BUSY:
	IF XpFeedback[i].sName.CallMoveX.Done THEN
		seqMoveXM[i]:=DONE;
	ELSIF Xpfeedback[i].sName.CallMoveX.Aborted THEN
		seqMoveXM[i]:=ABORT;
	ELSIF Xpfeedback[i].sName.CallMoveX.Error THEN	
		seqMoveXM[i]:=ERROR;
	END_IF

DONE:
	IF NOT MoveXM[i] THEN
	   seqMoveXM[i]:=READY;
	END_IF

ERROR:
	IF NOT MoveXM[i] THEN
	   seqMoveXM[i]:=READY;
	END_IF

ABORT:
	IF NOT MoveXM[i] THEN
	   seqMoveXM[i]:=READY;
	END_IF
	
END_CASE
END_ACTION

ACTION callMoveX_2m:
//MoveX2m
(*
	CASE seqMoveX_2m OF
		INIT:
        seqMoveX_2m:=READY;	
	 READY:
	 IF MoveX_2m THEN
	ConstraintXY[i].SetValuesVADJ(V:=velocity_xy[i] , A:=15000 , D:=15000 , J:=100000 );
	 
		Xpmover[i].MoveX(commandFeedback:=xpFeedback[i][14] , targetPosition:= positionTargetX[i] , refSys:=Xpmover[i].MCTOPLC.SET.PhysicalAreaID , 
         constraint:=ConstraintXY[i] );
		seqMoveX_2m:=BUSY;
		
		Xpmover[i].MoveX(commandFeedback:=xpFeedback[i][14], targetPosition:= positionTargetX[i] , refSys:=Xpmover[i].MCTOPLC.SET.PhysicalAreaID , 
         constraint:=ConstraintXY[i] );
		seqMoveX_2m:=BUSY;
		
		
		END_IF
		
		
		
   BUSY:
    IF  XpFeedback[0][14].Done THEN
		seqMoveX_2m:=DONE;
    ELSIF Xpfeedback[0][14].Aborted THEN
		seqMoveX_2m:=ABORT;
	ELSIF Xpfeedback[0][14].Error THEN	
		seqMoveX_2m:=ERROR;
	END_IF
		//
	
		DONE:
		IF NOT MoveX_2m THEN
	       seqMoveX_2m:=READY;
		END_IF
		
		ERROR:
		IF NOT MoveX_2m THEN
	       seqMoveX_2m:=READY;
		END_IF
		
		ABORT:
		IF NOT MoveX_2m THEN
	       seqMoveX_2m:=READY;
		END_IF
		
	END_CASE
	*)
END_ACTION

ACTION callMoveY:
CASE seqMoveYM[i] OF

INIT:
	seqMoveYM[i]:=READY;	

READY:
	IF MoveYM[i]THEN
		MoveYM[i] := FALSE;
		ConstraintXY[i].SetValuesVADJ(
			V:=velocity_xy[i] ,A:=15000 , D:=15000 , J:=100000 );
	 
		Xpmover[i].MoveY(
			commandFeedback:=xpFeedback[i].sName.CallMoveY,
			targetPosition:= positionTargetY[i],
			refSys:=Xpmover[i].MCTOPLC.SET.PhysicalAreaID, 
			constraint:=ConstraintXY[i] );
		seqMoveYM[i]:=BUSY;
	END_IF
	
BUSY:
	IF XpFeedback[i].sName.CallMoveY.Done THEN
		seqMoveYM[i]:=DONE;
	ELSIF Xpfeedback[i].sName.CallMoveY.Aborted THEN
		seqMoveYM[i]:=ABORT;
	ELSIF Xpfeedback[i].sName.CallMoveY.Error THEN	
		seqMoveYM[i]:=ERROR;
	END_IF

DONE:
	IF NOT MoveYM[i] THEN
	   seqMoveYM[i]:=READY;
	END_IF

ERROR:
	IF NOT MoveYM[i] THEN
	   seqMoveYM[i]:=READY;
	END_IF

ABORT:
	IF NOT MoveYM[i] THEN
	   seqMoveYM[i]:=READY;
	END_IF
	
END_CASE
END_ACTION

ACTION callMoveZ:
CASE seqMoveZM[i] OF

INIT:
	seqMoveZM[i]:=READY;
	Constratint_ZABC[i].SetLimit(
		Coordinate:= Coord_Mcs_A1, 
		V:= 100 , 
		A:= 100 , 
		D:= 100, 
		J:= 1000);
	
READY:
	IF moveZM[i]THEN
		MoveZM[i] := FALSE;	
		Constratint_ZABC[i].AddLimit(
			Coordinate:= Coord_Mcs_A1, 
			V:= 100 , 
			A:= 100 , 
			D:= 100, 
			J:= 1000);
		Xpmover[i].MoveZ(
			commandFeedback:=xpFeedback[i].sName.CallMoveZ , 
			targetPosition:=positionTargetZ[i] , 
			constraint:=ConstraTINT_zabc[i]);
		seqMoveZM[i]:=BUSY;
	END_IF
		
BUSY:
    IF XpFeedback[i].sName.CallMoveZ.Done THEN
		seqMoveZM[i]:=DONE;
    ELSIF Xpfeedback[i].sName.CallMoveZ.Aborted THEN
		seqMoveZM[i]:=ABORT;
	ELSIF Xpfeedback[i].sName.CallMoveZ.Error THEN	
		seqMoveZM[i]:=ERROR;
	END_IF
	
DONE:
	IF NOT MoveZM[i] THEN
	   seqMoveZM[i]:=READY;
	END_IF
	
ERROR:
	IF NOT MoveZM[i] THEN
	   seqMoveZM[i]:=READY;
	END_IF
	
ABORT:
	IF NOT MoveZM[i] THEN
	   seqMoveZM[i]:=READY;
	END_IF
		
END_CASE
END_ACTION

ACTION CallReset:
CASE seqResetM[i] OF
	
INIT:
	seqResetM[i]:=READY;

READY:
	IF ResetM[i]THEN
		Xpmover[i].Reset(commandFeedback:=XpFeedBack[i].sName.CallReset);
		seqResetM[i]:=BUSY;
	END_IF
		
BUSY:
	IF xpFeedback[i].sName.CallReset.Done THEN
		ResetM[i]:=FALSE;
		seqResetM[i]:=DONE;
	END_IF
		
DONE:
	IF NOT ResetM[i] THEN
		seqResetM[i]:=READY;
	END_IF

END_CASE
END_ACTION

ACTION seq_JoinTrack:
IF bJoinTrackseq THEN
	bJoinTrackseq := FALSE;
	
	FOR i:=0 TO gvl.MAX_MOVER DO
		ConstraintXY[i].SetValuesVADJ(V:=velocity_xy[i] , A:=15000 , D:=15000 , J:=100000 );
		velocity_xy[i] := 50;
	END_FOR
	
	Xpmover[0].JoinTrack(commandFeedback:= Xpfeedback[0].sName.SeqJoinTrack,
		targetTrack:= XpTrack[E_TrackName.Wait],
		constraint := ConstraintXY[0],
		options := 0);
		
	xpmover[1].JoinTrack(commandFeedback:= Xpfeedback[1].sName.SeqJoinTrack,
		targetTrack:= XpTrack[E_TrackName.EndA],
		constraint := ConstraintXY[1],
		options := 0);
END_IF

IF bMoveTrackSeq THEN
	bMoveTrackSeq := FALSE;
	fbStateTrack[0].bMoveState := TRUE;
	fbStateTrack[1].bMoveState := TRUE;
ELSE
	fbStateTrack[0].bMoveState := FALSE;
	fbStateTrack[1].bMoveState := FALSE;
END_IF

IF GVL.bfill THEN
	GVL.bfill  := FALSE;
END_IF

diCountSum := 0;
FOR i:=0 TO GVL.MAX_MOVER DO
	diCountSum := diCountSum + fbStateTrack[i].icount;
END_FOR

IF CountReset THEN
	CountReset := FALSE;
	FOR i:=0 TO GVL.MAX_MOVER DO
		fbStateTrack[i].breset := TRUE;
	END_FOR
END_IF
END_ACTION

ACTION update:
FOR i:=0 TO gvl.MAX_MOVER DO //xpmover 
	XpMover[i].update();
	FOR k:=0 TO MAX_FEEDBACK DO	
		Xpfeedback[i].aArray[k].Update();
	END_FOR
END_FOR

FOR t:=0 TO MAX_TRACK DO
    XpTrack[t].Update();
END_FOR
END_ACTION

END_PROGRAM

// ---- GlobalTextList.TcGTLO
TEXTLIST GlobalTextList
  582 = '%0,1f'
  833 = '%0.1f'
  192 = '%0.1f /s'
  27 = '%0.1f deg/s'
  12 = '%0.1f mm/s'
  142 = '%d'
  807 = '%S'
  450 = '1'
  857 = '2'
  13 = '22'
  974 = 'A'
  287 = 'A(Rx)'
  255 = 'B'
  85 = 'B(Ry)'
  421 = 'BFILL'
  484 = 'bstop'
  865 = 'C'
  567 = 'C(Rz)'
  424 = 'count'
  375 = 'disable'
  989 = 'Disable'
  74 = 'Enable'
  644 = 'Halt'
  595 = 'JoinTrack'
  973 = 'JoinTrack\nMover2台順次'
  117 = 'JoinTrack 1'
  83 = 'LeaveTrack'
  545 = 'moveA'
  66 = 'moveB'
  980 = 'moveC'
  981 = 'MoveOn'
  361 = 'MoveOnTrack'
  549 = 'MoveOnTrack 1'
  885 = 'Mover1'
  533 = 'Mover2'
  882 = 'Mover3'
  44 = 'Mover4'
  602 = 'MoverX1'
  542 = 'MoverX2'
  668 = 'MoveTrack\nMover2台同時'
  734 = 'movex'
  52 = 'movex1'
  608 = 'movey'
  742 = 'moveY'
  360 = 'moveY1'
  884 = 'moveZ'
  86 = 'Point to Move'
  994 = 'RealTime'
  474 = 'Reset'
  187 = 'reset'
  233 = 'Target Pos'
  977 = 'velo'
  587 = 'velocity_c'
  520 = 'velocity_xy'
  226 = 'X'
  493 = 'X1'
  377 = 'Y'
  645 = 'Y1'
  95 = 'Z'
  372 = '[0]'
  901 = '[0][0]'
  862 = '[1]'
END_TEXTLIST

// ---- VISUs/Visualization.TcVIS
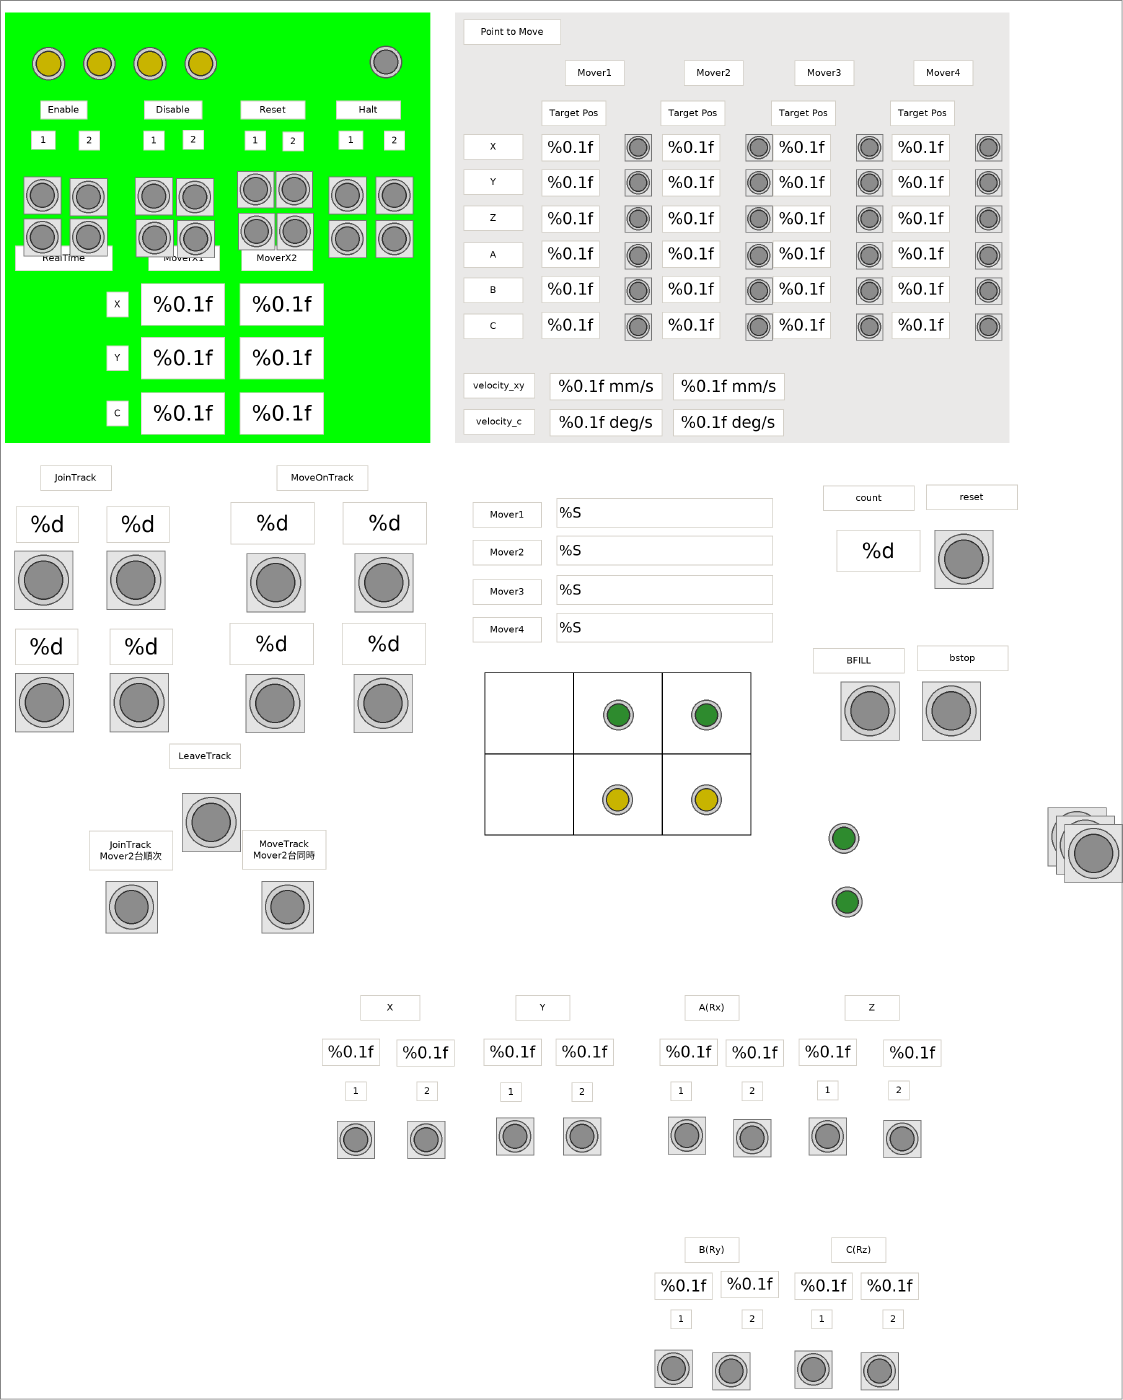
VISUALIZATION Visualization  // 1340x1670
    Rectangle (543,15 661x513)
    Rectangle (6,15 507x513)
    PushSwitch (161,194 45x80), tooltip "disable", variable: MAIN.disableM[0], behaviour: TAP, style: Switch-PushSwitch-Gray
    Lamp1 (35,43 46x66), variable: MAIN.bMoverEnable[0], style: Lamp-Lamp1-Yellow
    PushSwitchLed (402,1325 45x69), tooltip "movex", variable: MAIN.moveXM[0], behaviour: TOGGLE, style: Switch-PushSwitchLed-Gray
    Textfield (384,1239 69x32), "%0.1f", text variable: MAIN.positionTargetX[0]
        OnMouseClick: write the text variable via Default, min 60, max 660
    Textfield (430,1187 71x30), "X"
    Textfield (577,1239 69x32), "%0.1f", text variable: MAIN.positionTargetY[0]
        OnMouseClick: write the text variable via Default, min 60, max 420
    Textfield (615,1187 65x30), "Y"
    PushSwitchLed (592,1324 45x63), tooltip "moveY", variable: MAIN.moveYM[0], behaviour: TOGGLE, style: Switch-PushSwitchLed-Gray
    Textfield (553,445 85x30), "velocity_xy"
    Textfield (817,1187 65x30), "A(Rx)"
    Textfield (787,1239 69x32), "%0.1f", text variable: MAIN.positionTargetA[0]
        OnMouseClick: write the text variable via Default, min -5, max 5
    PushSwitchLed (797,1323 45x63), tooltip "moveA", variable: MAIN.moveAM[0], behaviour: TOGGLE, style: Switch-PushSwitchLed-Gray
    Textfield (817,1476 65x30), "B(Ry)"
    Textfield (781,1518 69x32), "%0.1f", text variable: MAIN.positionTargetB[0]
        OnMouseClick: write the text variable via Default, min -5, max 5
    PushSwitchLed (781,1598 45x69), tooltip "moveB", variable: MAIN.moveBM[0], behaviour: TOGGLE, style: Switch-PushSwitchLed-Gray
    Textfield (1008,1187 65x30), "Z"
    Textfield (953,1239 69x32), "%0.1f", text variable: MAIN.positionTargetZ[0]
        OnMouseClick: write the text variable via Default, min 2, max 5
    PushSwitchLed (965,1324 45x63), tooltip "moveZ", variable: MAIN.moveZM[0], behaviour: TOGGLE, style: Switch-PushSwitchLed-Gray
    Textfield (992,1476 65x30), "C(Rz)"
    Textfield (948,1518 69x32), "%0.1f", text variable: MAIN.positionTargetC[0]
        OnMouseClick: write the text variable via Default
    PushSwitchLed (948,1599 45x69), tooltip "moveC", variable: MAIN.moveCM[0], behaviour: TOGGLE, style: Switch-PushSwitchLed-Gray
    Textfield (553,488 85x30), "velocity_c"
    Textfield (168,338 100x50), "%0.1f", text variable: MAIN.Xpmover[0].MCTOPLC.ACT.ActPos.x
    Textfield (168,402 100x50), "%0.1f", text variable: MAIN.Xpmover[0].MCTOPLC.ACT.ActPos.y
    Textfield (168,468 100x50), "%0.1f", text variable: MAIN.Xpmover[0].MCTOPLC.ACT.ActPos.c
    Textfield (177,293 85x30), "MoverX1"
    PushSwitch (17,657 70x70), variable: MAIN.JoinTrack[0], behaviour: TOGGLE, style: Switch-PushSwitch-Gray
    PushSwitch (217,946 70x70), variable: MAIN.LeaveTrack[0], behaviour: TOGGLE, style: Switch-PushSwitch-Gray
    Textfield (48,555 85x30), "JoinTrack"
    Textfield (202,887 85x30), "LeaveTrack"
    Textfield (19,604 75x43), "%d", text variable: MAIN.numberTrack[0]
        OnMouseClick: write the text variable via Default, min 0
    PushSwitch (283,195 44x62), variable: MAIN.ResetM[0], invisible if: MAIN.ResetM, behaviour: TOGGLE, style: Switch-PushSwitch-Gray
    Textfield (48,120 56x22), "Enable"
    Textfield (172,120 69x22), "Disable"
    Textfield (287,120 77x22), "Reset"
    PushSwitch (392,193 45x80), variable: MAIN.HaltM[0], invisible if: MAIN.HaltM, behaviour: TOGGLE, style: Switch-PushSwitch-Gray
    Textfield (37,156 29x22), "1"
    Textfield (94,156 25x23), "2"
    Lamp1 (96,44 45x64), variable: MAIN.bMoverEnable[1], style: Lamp-Lamp1-Yellow
    Textfield (171,156 25x23), "1"
    Textfield (218,155 25x23), "2"
    PushSwitch (210,195 45x80), tooltip "disable", variable: MAIN.disableM[1], behaviour: TAP, style: Switch-PushSwitch-Gray
    Textfield (292,156 25x23), "1"
    PushSwitch (329,195 44x62), variable: MAIN.ResetM[1], invisible if: MAIN.ResetM, behaviour: TOGGLE, style: Switch-PushSwitch-Gray
    Textfield (337,157 25x23), "2"
    Textfield (497,1290 25x23), "2"
    Textfield (412,1290 25x23), "1"
    PushSwitchLed (486,1325 45x69), tooltip "movex", variable: MAIN.moveXM[1], behaviour: TOGGLE, style: Switch-PushSwitchLed-Gray
    Textfield (473,1240 69x32), "%0.1f", text variable: MAIN.positionTargetX[1]
        OnMouseClick: write the text variable via Default, min 60, max 660
    Textfield (663,1239 69x32), "%0.1f", text variable: MAIN.positionTargetY[1]
        OnMouseClick: write the text variable via Default, min 60, max 420
    PushSwitchLed (672,1324 45x63), tooltip "moveY", variable: MAIN.moveYM[1], behaviour: TOGGLE, style: Switch-PushSwitchLed-Gray
    Textfield (866,1240 69x32), "%0.1f", text variable: MAIN.positionTargetA[1]
        OnMouseClick: write the text variable via Default, min -5, max 5
    PushSwitchLed (875,1326 45x63), tooltip "moveA", variable: MAIN.moveAM[1], behaviour: TOGGLE, style: Switch-PushSwitchLed-Gray
    PushSwitchLed (1054,1327 45x63), tooltip "moveZ", variable: MAIN.moveZM[1], behaviour: TOGGLE, style: Switch-PushSwitchLed-Gray
    Textfield (1054,1240 69x32), "%0.1f", text variable: MAIN.positionTargetZ[1]
        OnMouseClick: write the text variable via Default, min 2, max 5
    PushSwitchLed (850,1601 45x69), tooltip "moveB", variable: MAIN.moveBM[1], behaviour: TOGGLE, style: Switch-PushSwitchLed-Gray
    Textfield (860,1516 69x32), "%0.1f", text variable: MAIN.positionTargetB[0]
        OnMouseClick: write the text variable via Default, min -5, max 5
    Textfield (1027,1518 69x32), "%0.1f", text variable: MAIN.positionTargetC[1]
        OnMouseClick: write the text variable via Default
    PushSwitchLed (1027,1601 45x69), tooltip "moveC", variable: MAIN.moveCM[1], behaviour: TOGGLE, style: Switch-PushSwitchLed-Gray
    Textfield (288,293 85x30), "MoverX2"
    Textfield (286,338 100x50), "%0.1f", text variable: MAIN.Xpmover[1].MCTOPLC.ACT.ActPos.x
    Textfield (286,402 100x50), "%0.1f", text variable: MAIN.Xpmover[1].MCTOPLC.ACT.ActPos.y
    Textfield (286,468 100x50), "%0.1f", text variable: MAIN.Xpmover[1].MCTOPLC.ACT.ActPos.c
    PushSwitch (448,193 45x80), variable: MAIN.HaltM[1], invisible if: MAIN.HaltM, behaviour: TOGGLE, style: Switch-PushSwitch-Gray
    Textfield (404,156 29x22), "1"
    Textfield (458,156 25x23), "2"
    Textfield (597,1291 25x23), "1"
    Textfield (682,1291 25x23), "2"
    Textfield (800,1290 25x23), "1"
    Textfield (885,1290 25x23), "2"
    Textfield (975,1289 25x23), "1"
    Textfield (1060,1289 25x23), "2"
    Textfield (800,1562 25x23), "1"
    Textfield (885,1562 25x23), "2"
    Textfield (968,1562 25x23), "1"
    Textfield (1053,1562 25x23), "2"
    Textfield (553,160 71x30), "X"
    Textfield (674,72 71x30), "Mover1"
    Textfield (646,160 69x32), "%0.1f", text variable: MAIN.positionTargetX[0]
        OnMouseClick: write the text variable via Default, min 60, max 660
    PushSwitch (731,160 61x32), variable: MAIN.moveXM[0], behaviour: TOGGLE, style: Switch-PushSwitch-Gray
    Textfield (553,202 71x30), "Y"
    Textfield (646,202 69x32), "%0.1f", text variable: MAIN.positionTargetY[0]
        OnMouseClick: write the text variable via Default, min 60, max 420
    PushSwitch (731,202 61x32), variable: MAIN.moveYM[0], behaviour: TOGGLE, style: Switch-PushSwitch-Gray
    Textfield (553,245 71x30), "Z"
    Textfield (646,245 69x32), "%0.1f", text variable: MAIN.positionTargetZ[0]
        OnMouseClick: write the text variable via Default, min 2, max 5
    PushSwitch (731,245 61x32), variable: MAIN.moveZM[0], behaviour: TOGGLE, style: Switch-PushSwitch-Gray
    Textfield (553,289 71x30), "A"
    PushSwitch (731,289 61x32), variable: MAIN.moveAM[0], behaviour: TOGGLE, style: Switch-PushSwitch-Gray
    Textfield (553,331 71x30), "B"
    PushSwitch (731,331 61x32), variable: MAIN.moveBM[0], behaviour: TOGGLE, style: Switch-PushSwitch-Gray
    Textfield (553,374 71x30), "C"
    PushSwitch (731,374 61x32), variable: MAIN.moveCM[0], behaviour: TOGGLE, style: Switch-PushSwitch-Gray
    Textfield (646,287 69x32), "%0.1f", text variable: MAIN.positionTargetA[0]
        OnMouseClick: write the text variable via Default, min -5, max 5
    Textfield (646,329 69x32), "%0.1f", text variable: MAIN.positionTargetB[0]
        OnMouseClick: write the text variable via Default, min -5, max 5
    Textfield (646,372 69x32), "%0.1f", text variable: MAIN.positionTargetC[0]
        OnMouseClick: write the text variable via Default
    Textfield (816,72 71x30), "Mover2"
    Textfield (790,160 69x32), "%0.1f", text variable: MAIN.positionTargetX[1]
        OnMouseClick: write the text variable via Default, min 60, max 660
    PushSwitch (875,160 61x32), variable: MAIN.moveXM[1], behaviour: TOGGLE, style: Switch-PushSwitch-Gray
    Textfield (790,202 69x32), "%0.1f", text variable: MAIN.positionTargetY[1]
        OnMouseClick: write the text variable via Default, min 60, max 420
    PushSwitch (875,202 61x32), variable: MAIN.moveYM[1], behaviour: TOGGLE, style: Switch-PushSwitch-Gray
    Textfield (790,245 69x32), "%0.1f", text variable: MAIN.positionTargetZ[1]
        OnMouseClick: write the text variable via Default, min 2, max 5
    PushSwitch (875,245 61x32), variable: MAIN.moveZM[1], behaviour: TOGGLE, style: Switch-PushSwitch-Gray
    PushSwitch (875,289 61x32), variable: MAIN.moveAM[1], behaviour: TOGGLE, style: Switch-PushSwitch-Gray
    PushSwitch (875,331 61x32), variable: MAIN.moveBM[1], behaviour: TOGGLE, style: Switch-PushSwitch-Gray
    PushSwitch (875,374 61x32), variable: MAIN.moveCM[1], behaviour: TOGGLE, style: Switch-PushSwitch-Gray
    Textfield (790,287 69x32), "%0.1f", text variable: MAIN.positionTargetA[1]
        OnMouseClick: write the text variable via Default, min -5, max 5
    Textfield (790,329 69x32), "%0.1f", text variable: MAIN.positionTargetB[1]
        OnMouseClick: write the text variable via Default, min -5, max 5
    Textfield (790,372 69x32), "%0.1f", text variable: MAIN.positionTargetC[1]
        OnMouseClick: write the text variable via Default
    Textfield (646,120 77x30), "Target Pos"
    Textfield (788,120 77x30), "Target Pos"
    Textfield (553,23 116x30), "Point to Move"
    Textfield (127,348 26x30), "X"
    Textfield (127,412 26x30), "Y"
    Textfield (127,478 26x30), "C"
    Textfield (401,120 77x22), "Halt"
    Textfield (18,293 116x30), "RealTime"
    Textfield (803,445 133x32), "%0.1f mm/s", text variable: MAIN.velocity_xy[1]
        OnMouseClick: write the text variable via Default
    Textfield (656,445 134x32), "%0.1f mm/s", text variable: MAIN.velocity_xy[0]
        OnMouseClick: write the text variable via Default
    Textfield (656,488 134x32), "%0.1f deg/s", text variable: MAIN.velocity_c[0]
        OnMouseClick: write the text variable via Default
    Textfield (803,488 132x32), "%0.1f deg/s", text variable: MAIN.velocity_c[1]
        OnMouseClick: write the text variable via Default
    PushSwitch (28,193 45x80), tooltip "Enable", variable: MAIN.enableM[0], behaviour: TAP, style: Switch-PushSwitch-Gray
    PushSwitch (83,195 45x80), tooltip "Enable", variable: MAIN.enableM[1], behaviour: TAP, style: Switch-PushSwitch-Gray
    PushSwitch (294,660 70x70), variable: MAIN.fbStateTrack[0].bMoveState, behaviour: TOGGLE, style: Switch-PushSwitch-Gray
    Textfield (275,599 100x50), "%d", text variable: MAIN.fbStateTrack[0].iStateTrack
    PushSwitch (423,660 70x70), variable: MAIN.fbStateTrack[1].bMoveState, behaviour: TOGGLE, style: Switch-PushSwitch-Gray
    Textfield (409,599 100x50), "%d", text variable: MAIN.fbStateTrack[1].iStateTrack
    PushSwitch (127,657 70x70), variable: MAIN.JoinTrack[1], behaviour: TOGGLE, style: Switch-PushSwitch-Gray
    Group (578,802 318x194)
        Rectangle (0,0 106x97)
        Rectangle (0,97 106x97)
        Rectangle (106,0 106x97)
        Rectangle (106,97 106x97)
        Rectangle (212,0 106x97)
        Rectangle (212,97 106x97)
    Lamp1 (715,933 44x42), variable: GVL.bBusyB, style: Lamp-Lamp1-Yellow
    Lamp1 (821,933 44x42), variable: GVL.bBusyA, style: Lamp-Lamp1-Yellow
    Textfield (664,594 258x35), "%S", text list: 'TextList_TrackState', text index: MAIN.fbStateTrack[0].iStateTrack
    Textfield (664,639 258x35), "%S", text list: 'TextList_TrackState', text index: MAIN.fbStateTrack[1].iStateTrack
    Textfield (564,599 82x30), "Mover1"
    Textfield (564,644 82x30), "Mover2"
    PushSwitch (126,1047 62x70), variable: MAIN.bJoinTrackseq, behaviour: TOGGLE, style: Switch-PushSwitch-Gray
    Textfield (106,991 100x47), "JoinTrack Mover2台順次"
    PushSwitch (312,1047 62x70), variable: MAIN.bJoinTrackseq, behaviour: TOGGLE, style: Switch-PushSwitch-Gray
    Textfield (289,990 100x47), "MoveTrack Mover2台同時"
    Textfield (330,555 109x30), "MoveOnTrack"
    Lamp1 (821,832 44x42), variable: GVL.bDoneA, style: Lamp-Lamp1-Green
    Lamp1 (716,832 44x42), variable: GVL.bDoneB, style: Lamp-Lamp1-Green
    PushSwitch (1003,813 70x70), variable: GVL.bfill, behaviour: TOGGLE, style: Switch-PushSwitch-Gray
    Textfield (970,773 109x30), "BFILL"
    Lamp1 (985,979 44x42), variable: MAIN.fbStateTrack[0].bGoAline, style: Lamp-Lamp1-Green
    Lamp1 (989,1055 44x42), variable: MAIN.fbStateTrack[1].bGoAline, style: Lamp-Lamp1-Green
    PushSwitch (1100,813 70x70), variable: GVL.bstop, behaviour: TOGGLE, style: Switch-PushSwitch-Gray
    Textfield (1094,770 109x30), "bstop"
    Textfield (998,632 100x50), "%d", text variable: MAIN.diCountSum
    Textfield (982,579 109x30), "count"
    PushSwitch (1250,963 70x70), variable: GVL.bstop, behaviour: TOGGLE, style: Switch-PushSwitch-Gray
    PushSwitch (1260,973 70x70), variable: GVL.bstop, behaviour: TOGGLE, style: Switch-PushSwitch-Gray
    PushSwitch (1270,983 70x70), variable: GVL.bstop, behaviour: TOGGLE, style: Switch-PushSwitch-Gray
    PushSwitch (1115,632 70x70), variable: MAIN.CountReset, behaviour: TOGGLE, style: Switch-PushSwitch-Gray
    Textfield (1105,578 109x30), "reset"
    PushSwitch (28,243 45x80), tooltip "Enable", variable: MAIN.enableM[2], behaviour: TAP, style: Switch-PushSwitch-Gray
    PushSwitch (83,243 45x80), tooltip "Enable", variable: MAIN.enableM[3], behaviour: TAP, style: Switch-PushSwitch-Gray
    PushSwitch (162,244 45x80), tooltip "disable", variable: MAIN.disableM[2], behaviour: TAP, style: Switch-PushSwitch-Gray
    PushSwitch (211,245 45x80), tooltip "disable", variable: MAIN.disableM[3], behaviour: TAP, style: Switch-PushSwitch-Gray
    PushSwitch (284,245 44x62), variable: MAIN.ResetM[2], invisible if: MAIN.ResetM, behaviour: TOGGLE, style: Switch-PushSwitch-Gray
    PushSwitch (330,245 44x62), variable: MAIN.ResetM[3], invisible if: MAIN.ResetM, behaviour: TOGGLE, style: Switch-PushSwitch-Gray
    PushSwitch (448,245 45x80), variable: MAIN.HaltM[3], invisible if: MAIN.HaltM, behaviour: TOGGLE, style: Switch-PushSwitch-Gray
    PushSwitch (392,245 45x80), variable: MAIN.HaltM[2], invisible if: MAIN.HaltM, behaviour: TOGGLE, style: Switch-PushSwitch-Gray
    Textfield (948,72 71x30), "Mover3"
    Textfield (922,160 69x32), "%0.1f", text variable: MAIN.positionTargetX[2]
        OnMouseClick: write the text variable via Default, min 60, max 660
    PushSwitch (1007,160 61x32), variable: MAIN.moveXM[2], behaviour: TOGGLE, style: Switch-PushSwitch-Gray
    Textfield (922,202 69x32), "%0.1f", text variable: MAIN.positionTargetY[2]
        OnMouseClick: write the text variable via Default, min 60, max 420
    PushSwitch (1007,202 61x32), variable: MAIN.moveYM[2], behaviour: TOGGLE, style: Switch-PushSwitch-Gray
    Textfield (922,245 69x32), "%0.1f", text variable: MAIN.positionTargetZ[2]
        OnMouseClick: write the text variable via Default, min 2, max 5
    PushSwitch (1007,245 61x32), variable: MAIN.moveZM[2], behaviour: TOGGLE, style: Switch-PushSwitch-Gray
    PushSwitch (1007,289 61x32), variable: MAIN.moveAM[2], behaviour: TOGGLE, style: Switch-PushSwitch-Gray
    PushSwitch (1007,331 61x32), variable: MAIN.moveBM[2], behaviour: TOGGLE, style: Switch-PushSwitch-Gray
    PushSwitch (1007,374 61x32), variable: MAIN.moveCM[2], behaviour: TOGGLE, style: Switch-PushSwitch-Gray
    Textfield (922,287 69x32), "%0.1f", text variable: MAIN.positionTargetA[2]
        OnMouseClick: write the text variable via Default, min -5, max 5
    Textfield (922,329 69x32), "%0.1f", text variable: MAIN.positionTargetB[2]
        OnMouseClick: write the text variable via Default, min -5, max 5
    Textfield (922,372 69x32), "%0.1f", text variable: MAIN.positionTargetC[2]
        OnMouseClick: write the text variable via Default
    Textfield (920,120 77x30), "Target Pos"
    Textfield (1090,72 71x30), "Mover4"
    Textfield (1064,160 69x32), "%0.1f", text variable: MAIN.positionTargetX[3]
        OnMouseClick: write the text variable via Default, min 60, max 660
    PushSwitch (1149,160 61x32), variable: MAIN.moveXM[3], behaviour: TOGGLE, style: Switch-PushSwitch-Gray
    Textfield (1064,202 69x32), "%0.1f", text variable: MAIN.positionTargetY[3]
        OnMouseClick: write the text variable via Default, min 60, max 420
    PushSwitch (1149,202 61x32), variable: MAIN.moveYM[3], behaviour: TOGGLE, style: Switch-PushSwitch-Gray
    Textfield (1064,245 69x32), "%0.1f", text variable: MAIN.positionTargetZ[3]
        OnMouseClick: write the text variable via Default, min 2, max 5
    PushSwitch (1149,245 61x32), variable: MAIN.moveZM[3], behaviour: TOGGLE, style: Switch-PushSwitch-Gray
    PushSwitch (1149,289 61x32), variable: MAIN.moveAM[3], behaviour: TOGGLE, style: Switch-PushSwitch-Gray
    PushSwitch (1149,331 61x32), variable: MAIN.moveBM[3], behaviour: TOGGLE, style: Switch-PushSwitch-Gray
    PushSwitch (1149,374 61x32), variable: MAIN.moveCM[3], behaviour: TOGGLE, style: Switch-PushSwitch-Gray
    Textfield (1064,287 69x32), "%0.1f", text variable: MAIN.positionTargetA[3]
        OnMouseClick: write the text variable via Default, min -5, max 5
    Textfield (1064,329 69x32), "%0.1f", text variable: MAIN.positionTargetB[3]
        OnMouseClick: write the text variable via Default, min -5, max 5
    Textfield (1064,372 69x32), "%0.1f", text variable: MAIN.positionTargetC[3]
        OnMouseClick: write the text variable via Default
    Textfield (1062,120 77x30), "Target Pos"
    Textfield (127,604 75x43), "%d", text variable: MAIN.numberTrack[1]
        OnMouseClick: write the text variable via Default, min 0
    Textfield (18,750 75x43), "%d", text variable: MAIN.numberTrack[2]
        OnMouseClick: write the text variable via Default, min 0
    PushSwitch (18,803 70x70), variable: MAIN.JoinTrack[2], behaviour: TOGGLE, style: Switch-PushSwitch-Gray
    Textfield (131,750 75x43), "%d", text variable: MAIN.numberTrack[3]
        OnMouseClick: write the text variable via Default, min 0
    PushSwitch (131,803 70x70), variable: MAIN.JoinTrack[3], behaviour: TOGGLE, style: Switch-PushSwitch-Gray
    Textfield (274,743 100x50), "%d", text variable: MAIN.fbStateTrack[2].iStateTrack
    PushSwitch (293,804 70x70), variable: MAIN.fbStateTrack[2].bMoveState, behaviour: TOGGLE, style: Switch-PushSwitch-Gray
    PushSwitch (422,804 70x70), variable: MAIN.fbStateTrack[3].bMoveState, behaviour: TOGGLE, style: Switch-PushSwitch-Gray
    Textfield (408,743 100x50), "%d", text variable: MAIN.fbStateTrack[3].iStateTrack
    Textfield (564,691 82x30), "Mover3"
    Textfield (664,686 258x35), "%S", text list: 'TextList_TrackState', text index: MAIN.fbStateTrack[2].iStateTrack
    Textfield (664,731 258x35), "%S", text list: 'TextList_TrackState', text index: MAIN.fbStateTrack[3].iStateTrack
    Textfield (564,736 82x30), "Mover4"
    Lamp1 (156,43 46x66), variable: MAIN.bMoverEnable[2], style: Lamp-Lamp1-Yellow
    Lamp1 (217,44 45x64), variable: MAIN.bMoverEnable[3], style: Lamp-Lamp1-Yellow
    Lamp1 (438,42 45x64), variable: MAIN.bSlowStop, style: Lamp-Lamp1-Gray
END_VISUALIZATION
